{attribute 'GeneratedUsingTerminal: EJ9400-0000-0000'}
{attribute addProperty BoxType "EJ9400-0000-0000"}
{attribute addProperty Description "EJ9400-0000 Power supply module 2,5A"}
{attribute addProperty Physics "KK"}
{attribute addProperty Id "EJ9400"}
{attribute addProperty CRC "3037274076"}
{attribute addProperty Size "0"}
TYPE EJ9400_B5091FDC EXTENDS EtcSlaveTerminalBase_947E5A46 :
STRUCT
END_STRUCT
END_TYPE

(* stored: Version 1.2.0.0, ProductVersion 3.1.4024.11
   DUT EJ9400_B5091FDC: Id {60f906d6-ca1b-4250-ac37-8c352a89b1e3} *)
